{attribute 'GeneratedUsingTerminal: EK1122-0000-0018'}
{attribute addProperty BoxType "EK1122-0000-0018"}
{attribute addProperty Id "Beckhoff_EPP9xxxsub_EK1100EK1100_1FC0878B2A_0001_EPP9001_0060_0016EPP9001_1FC0878B2A_0002_EPP9001_0060_0017EPP9001_1FC0878B2A_0003_EPP9022_0060_0017EPP9022_32A9C19F48A_0004_EPP9022_9060_0017EPP9022_32A9C19F48"}
{attribute addProperty CRC "3073232419"}
{attribute addProperty Size "102"}
TYPE Beckhoff_EPP9xxxEK1122_B72DCE23 EXTENDS EK1122_1FC0878B :
STRUCT
	{attribute addProperty Name "Beckhoff_EPP9xxxsub_EK1100"}
	Beckhoff_EPP9xxxsub_EK1100 : EK1100_1FC0878B;
	{attribute addProperty Name "A_0001_EPP9001_0060_0016"}
	A_0001_EPP9001_0060_0016 : EPP9001_1FC0878B;
	{attribute addProperty Name "A_0002_EPP9001_0060_0017"}
	A_0002_EPP9001_0060_0017 : EPP9001_1FC0878B;
	{attribute addProperty Name "A_0003_EPP9022_0060_0017"}
	A_0003_EPP9022_0060_0017 : EPP9022_32A9C19F;
	{attribute addProperty Name "A_0004_EPP9022_9060_0017"}
	A_0004_EPP9022_9060_0017 : EPP9022_32A9C19F;
END_STRUCT
END_TYPE

(* stored: Version 1.2.0.0, ProductVersion 3.1.4024.9
   DUT Beckhoff_EPP9xxxEK1122_B72DCE23: Id {4a7ac678-e6d3-40e8-948f-96f4216780a6} *)
